SUBAPPLICATION SoftKeyT_PC_A_OPC_Adapter (* Geraet A (Station 11, 192.168.1.11): wie Softkey_Toggle_RPC_TO_Remote_BG_OPC, aber HMI (SoftKey + GreenWhiteBackground) und OPC-UA-Trigger sind getrennt - SoftKeyT_AE_AX buendelt die HMI hinter einem AE_AX-Plug, AE_AX_CLIENT_0_SUBSCRIBE_1 buendelt CLIENT_0 + AX_SUBSCRIBE_1 hinter einem AE_AX-Socket - 'SUB style': das Protokoll steckt im MyLib::sys-Composite, nicht in der Resource des Geraets *)
  (* Standard: 61499-2; Description: Copyright (c) 2026 Meisterschulen am Ostbahnhof This program and the accompanying materials are made available under the terms of the Eclipse Public License 2.0 which is available at https://www.eclipse.org/legal/epl-2.0/ SPDX-License-Identifier: EPL-2.0 *)
  (* Version 1.0, 2026-09-04, Franz Höpfinger, Meisterschulen am Ostbahnhof, initial API and implementation and/or initial documentation *)
  PACKAGE MyLib::sys;
  IMPORT isobus::UT::Q::const::IDs::ID_NULL;
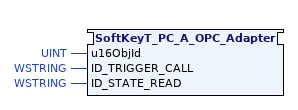
  VAR_INPUT
    u16ObjId : UINT := ID_NULL; (* Object ID Softkey/Background *)
    ID_TRIGGER_CALL : WSTRING; (* Remote-Methodenadresse (ACTION=CALL_METHOD) fuer den argumentlosen Trigger-Methodenaufruf auf Geraet B *)
    ID_STATE_READ : WSTRING; (* Lokal ueberwachte Adresse (BOOL, ACTION=READ) fuer den Flipflop-Zustand, wird von Geraet B remote beschrieben *)
  END_VAR
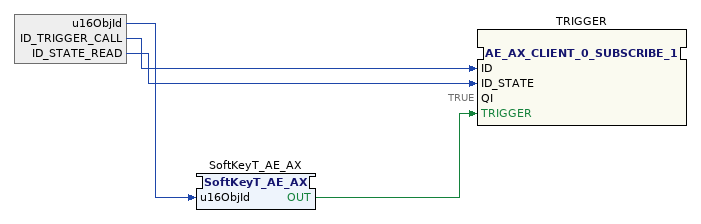
  FBS
    TRIGGER : adapter::net::AE_AX_CLIENT_0_SUBSCRIBE_1(QI := TRUE);
  END_FBS
  SUBAPPS
    SoftKeyT_AE_AX : MyLib::sys::SoftKeyT_AE_AX;
  END_SUBAPPS
  DATA_CONNECTIONS
    ID_TRIGGER_CALL TO TRIGGER.ID;
    ID_STATE_READ TO TRIGGER.ID_STATE;
    u16ObjId TO SoftKeyT_AE_AX.u16ObjId;
  END_CONNECTIONS
  ADAPTER_CONNECTIONS
    SoftKeyT_AE_AX.OUT TO TRIGGER.TRIGGER;
  END_CONNECTIONS
END_SUBAPPLICATION
